SYSTEM IncorrectParserTest1
  (* Version 1.0, 2025-07-22, dakudryashev *)
  APPLICATION IncorrectParserTest1App
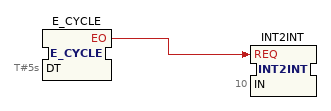
    FBS
      E_CYCLE : E_CYCLE(DT := T#5s);
      INT2INT : INT2INT(IN := 10);
    END_FBS
    EVENT_CONNECTIONS
      E_CYCLE.EO TO INT2INT.REQ;
    END_CONNECTIONS
  END_APPLICATION
  DEVICE FORTE_PC : FORTE_PC(MGR_ID := "localhost:61499" (* Device manager socket ID *))
    {SET_ATTRIBUTE(Profile, HOLOBLOC)}
    RESOURCE EMB_RES : EMB_RES
      EVENT_CONNECTIONS
        START.COLD TO IncorrectParserTest1App.E_CYCLE.START;
      END_CONNECTIONS
    END_RESOURCE
  END_DEVICE
  MAPPINGS
    IncorrectParserTest1App.E_CYCLE ON FORTE_PC.EMB_RES;
    IncorrectParserTest1App.INT2INT ON FORTE_PC.EMB_RES;
  END_MAPPINGS
  SEGMENTS
    Ethernet : Ethernet;
  END_SEGMENTS
  LINKS
    FORTE_PC => Ethernet;
  END_LINKS
END_SYSTEM
